TYPE ST_TTS_EPT :
STRUCT
	// TTS State
	eTTS: E_EPT;
	// TTS moduel state
	arrTTSLane: ARRAY [1..3] OF E_EPT;
END_STRUCT
END_TYPE

(* stored: Version 1.1.0.1, ProductVersion 3.1.4022.12
   DUT ST_TTS_EPT: Id {9ac28038-5b7a-41fd-987c-d5264f04a5e0} *)
